FUNCTION TryConvert_LREAL_TO_LREAL : BOOL
VAR_INPUT
	in : LREAL;
	out : REFERENCE TO LREAL;
END_VAR

out := in;
TryConvert_LREAL_TO_LREAL := TRUE;

END_FUNCTION

(* stored: Version 1.1.0.1, ProductVersion 3.1.4024.12
   POU TryConvert_LREAL_TO_LREAL: Id {9b39c0dc-9db2-4be3-b785-83f56fbb9881}, SpecialFunc None *)
